Universal Robots PolyScope program: Demo TiFa 10-01-2024.urp

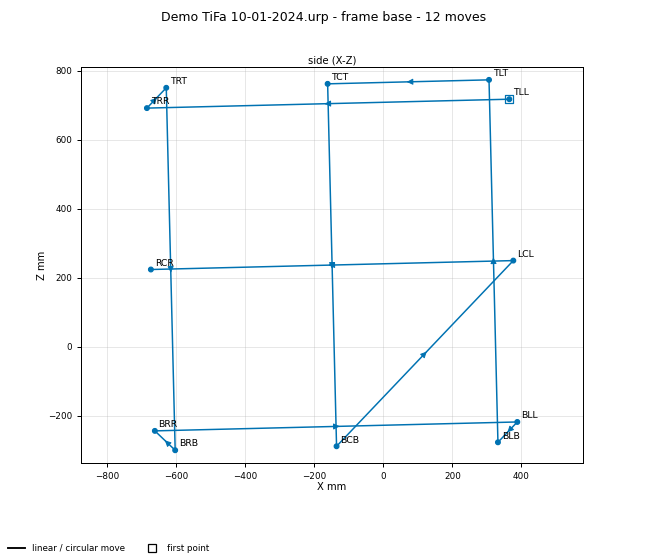
[picture p0: tool path of Demo TiFa 10-01-2024.urp in frame base, 12 of 12 moves have a stored position in this frame; points joined in program order, loops and branches not executed]
Program Demo TiFa 10-01-2024 (installation=Demo TiFa directory=/programs/usbdisk createdIn=5.13.0 lastSavedIn=5.13.0 robotSerialNumber=20225205328)
Calibrated DH parameters: a=[0.000015, -0.554412, -0.55278, -0.000048, 0.000048, 0]; d=[0.180794, 388.593069, -422.981807, 34.562793, 0.119661, 0.115558]; alpha=[1.570377, 0.000668, 0.00417, 1.56893, -1.569746, 0]; deltaTheta=[0, 0.437754, -0.691593, 0.253842, 0.000001, 0]
InitVariablesNode
Robot Program (runOnlyOnce=false)
  SuppressedNode
    Folder Define CC
      MoveL speed 250 mm/s, acceleration 1200 mm/s^2 (useActiveTCP=true) feature=Kozijn_Demo
        Waypoint CC: TCP in base x=-148.228 y=-773.929 z=236.857 mm, rx=0.6949 ry=-1.7899 rz=1.7889 rad; joints [-87.227, -128.672, -122.692, 71.274, 87.03, -42.484] deg; TCP offset x=0.884 y=1.376 z=84.755 mm, rx=0 ry=0 rz=0 rad; feature pose in base x=-149.69 y=-973.92 z=236.77 mm, rx=-1.2026 ry=-1.2236 rz=-1.2329 rad
  Folder Full circle 0deg
    MoveL speed 250 mm/s, acceleration 1200 mm/s^2 (useActiveTCP=true) feature=Kozijn_Demo
      Waypoint TLL: TCP in base x=365.055 y=-777.862 z=717.153 mm, rx=1.582 ry=-0.0318 rz=0.007 rad; joints [-42.763, -101.228, -97.529, 17.558, 41.783, -132.625] deg; TCP offset x=0.88 y=1.38 z=84.75 mm, rx=0 ry=0 rz=-0.7854 rad
      Waypoint TRR: TCP in base x=-684.539 y=-770.15 z=691.364 mm, rx=1.5759 ry=-0.0293 rz=0.0094 rad; joints [-128.821, -121.003, -72.672, 13.308, 128.022, -133.714] deg
      Waypoint TRT: TCP in base x=-628.471 y=-770.618 z=750.202 mm, rx=1.1999 ry=-1.2326 rz=1.2229 rad; joints [-125.847, -115.752, -74.413, 9.786, 125.657, -43.699] deg
      Waypoint BRB: TCP in base x=-602.658 y=-770.359 z=-299.466 mm, rx=1.1999 ry=-1.2327 rz=1.2229 rad; joints [-124.325, -185.934, -63.691, 69.144, 123.968, -43.876] deg
      Waypoint BRR: TCP in base x=-661.532 y=-769.998 z=-243.364 mm, rx=1.5759 ry=-0.0293 rz=0.0094 rad; joints [-127.581, -182.468, -62.696, 64.699, 126.638, -133.874] deg
      Waypoint BLL: TCP in base x=388.109 y=-777.678 z=-217.553 mm, rx=1.576 ry=-0.0293 rz=0.0094 rad; joints [-41.391, -175.41, -88.229, 83.165, 40.452, -133.284] deg
      Waypoint BLB: TCP in base x=332.05 y=-777.231 z=-276.466 mm, rx=1.1999 ry=-1.2327 rz=1.2229 rad; joints [-44.737, -180.477, -86.549, 86.566, 44.39, -43.327] deg
      Waypoint TLT: TCP in base x=306.211 y=-777.455 z=773.195 mm, rx=1.1999 ry=-1.2327 rz=1.2229 rad; joints [-46.493, -96.951, -96.622, 12.926, 46.289, -43.055] deg
  Folder Cross 0deg
    MoveL speed 250 mm/s, acceleration 1200 mm/s^2 (useActiveTCP=true) feature=Kozijn_Demo
      Waypoint TCT: TCP in base x=-161.147 y=-774.056 z=761.659 mm, rx=1.1999 ry=-1.2327 rz=1.2228 rad; joints [-88.529, -91.615, -103.59, 14.808, 88.314, -43.468] deg
      Waypoint BCB: TCP in base x=-135.312 y=-773.794 z=-287.963 mm, rx=1.1999 ry=-1.2327 rz=1.2228 rad; joints [-85.817, -181.687, -93.448, 94.755, 85.473, -43.687] deg
      Waypoint LCL: TCP in base x=376.597 y=-777.754 z=249.787 mm, rx=1.5759 ry=-0.0293 rz=0.0094 rad; joints [-42.085, -131.69, -111.247, 62.402, 41.167, -133.202] deg
      Waypoint RCR: TCP in base x=-673.018 y=-770.067 z=223.95 mm, rx=1.5759 ry=-0.0293 rz=0.0094 rad; joints [-128.204, -143.882, -86.243, 49.691, 127.298, -133.824] deg
  SuppressedNode
    Folder Inner circle BR 45deg
      MoveL speed 250 mm/s, acceleration 1200 mm/s^2 (useActiveTCP=true) feature=Kozijn_Demo
        Waypoint circBR_TR: TCP in base x=-481.193 y=-912.42 z=87.568 mm, rx=0.7529 ry=-0.3331 rz=-0.7421 rad; joints [-103.674, -146.065, -94.41, -70.561, 293.087, -337.663] deg
